// TIA Portal V17 export
// export: Created 2024-08-26T21:10:48.0587448Z, ExportSetting WithDefaults, DisplayName Totally Integrated Automation Portal, DisplayVersion V17 Update 7, DisplayName TIA Portal Openness, DisplayVersion V17 Update 7, DisplayName TIA Portal Version Control Interface, DisplayVersion V17, DisplayName SINAMICS Startdrive Advanced, DisplayVersion V17 SP2, DisplayName SINAMICS Startdrive G110M, G120, G120C, G120D, G120P, G115D, DisplayVersion V17 SP2, DisplayName SINAMICS Startdrive G130, G150, S120, S150, SINAMICS MV, S210, DisplayVersion V17 SP2, DisplayName STEP 7 Professional, DisplayVersion V17 Update 7, DisplayName STEP 7 Safety, DisplayVersion V17 Update 6, DisplayName WinCC Advanced / Unified PC, DisplayVersion V17 Update 7
FUNCTION "outputsMapping" : Void   // FC8, LAD
{ S7_Optimized_Access := 'TRUE' }
VERSION : 0.1
// stored: AutoNumber true, IsIECCheckEnabled false, SetENOAutomatically false, UDAEnableTagReadback false
BEGIN

REGION Network 1: OUTPUT VALVE ACTIVATION
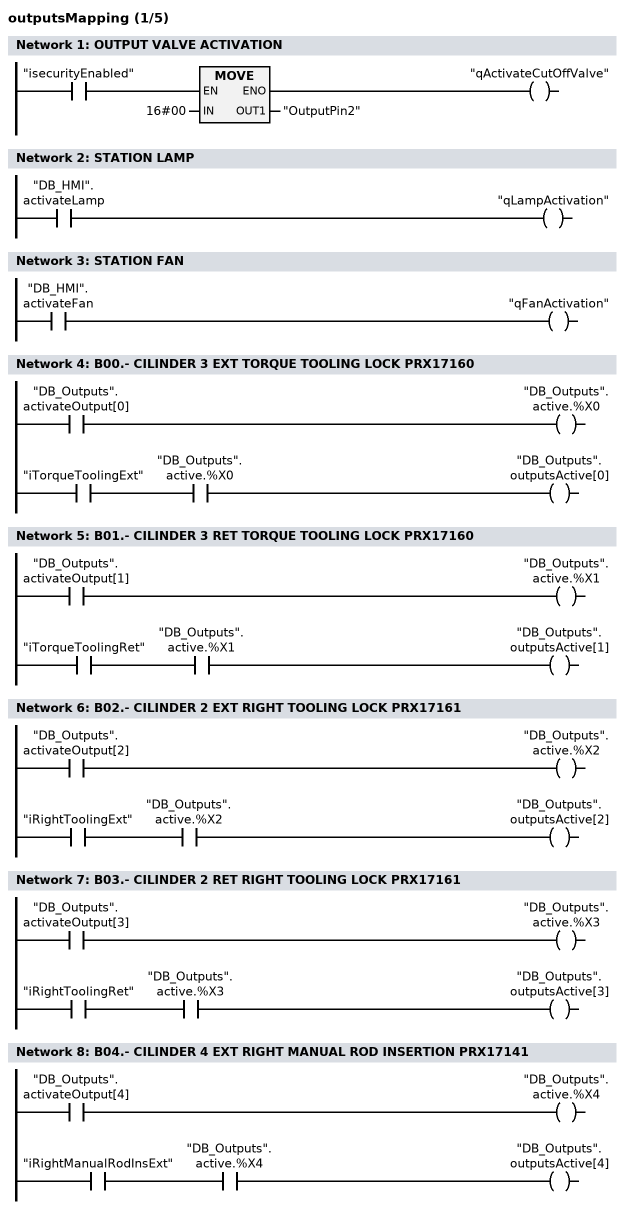
   RUNG wire#powerrail
      Contact( "isecurityEnabled" )
      Move(in := 16#00, out1 => "OutputPin2")
      Coil( "qActivateCutOffValve" )
   END_RUNG
   // the same network as SCL:
   IF "isecurityEnabled" THEN "OutputPin2" := 16#00; END_IF;
   "qActivateCutOffValve" := "isecurityEnabled";
END_REGION

REGION Network 2: STATION LAMP
   RUNG wire#powerrail
      Contact( "DB_HMI".activateLamp )
      Coil( "qLampActivation" )
   END_RUNG
   // the same network as SCL:
   "qLampActivation" := "DB_HMI".activateLamp;
END_REGION

REGION Network 3: STATION FAN
   RUNG wire#powerrail
      Contact( "DB_HMI".activateFan )
      Coil( "qFanActivation" )
   END_RUNG
   // the same network as SCL:
   "qFanActivation" := "DB_HMI".activateFan;
END_REGION

REGION Network 4: B00.- CILINDER 3 EXT TORQUE TOOLING LOCK PRX17160
   RUNG wire#powerrail
      Contact( "DB_Outputs".activateOutput[0] )
      Coil( "DB_Outputs".active.%X0 )
   END_RUNG
   RUNG wire#powerrail
      Contact( "iTorqueToolingExt" )
      Contact( "DB_Outputs".active.%X0 )
      Coil( "DB_Outputs".outputsActive[0] )
   END_RUNG
   // the same network as SCL:
   "DB_Outputs".active.%X0 := "DB_Outputs".activateOutput[0];
   "DB_Outputs".outputsActive[0] := "iTorqueToolingExt" AND "DB_Outputs".active.%X0;
END_REGION

REGION Network 5: B01.- CILINDER 3 RET TORQUE TOOLING LOCK PRX17160
   RUNG wire#powerrail
      Contact( "DB_Outputs".activateOutput[1] )
      Coil( "DB_Outputs".active.%X1 )
   END_RUNG
   RUNG wire#powerrail
      Contact( "iTorqueToolingRet" )
      Contact( "DB_Outputs".active.%X1 )
      Coil( "DB_Outputs".outputsActive[1] )
   END_RUNG
   // the same network as SCL:
   "DB_Outputs".active.%X1 := "DB_Outputs".activateOutput[1];
   "DB_Outputs".outputsActive[1] := "iTorqueToolingRet" AND "DB_Outputs".active.%X1;
END_REGION

REGION Network 6: B02.- CILINDER 2 EXT RIGHT TOOLING LOCK PRX17161
   RUNG wire#powerrail
      Contact( "DB_Outputs".activateOutput[2] )
      Coil( "DB_Outputs".active.%X2 )
   END_RUNG
   RUNG wire#powerrail
      Contact( "iRightToolingExt" )
      Contact( "DB_Outputs".active.%X2 )
      Coil( "DB_Outputs".outputsActive[2] )
   END_RUNG
   // the same network as SCL:
   "DB_Outputs".active.%X2 := "DB_Outputs".activateOutput[2];
   "DB_Outputs".outputsActive[2] := "iRightToolingExt" AND "DB_Outputs".active.%X2;
END_REGION

REGION Network 7: B03.- CILINDER 2 RET RIGHT TOOLING LOCK PRX17161
   RUNG wire#powerrail
      Contact( "DB_Outputs".activateOutput[3] )
      Coil( "DB_Outputs".active.%X3 )
   END_RUNG
   RUNG wire#powerrail
      Contact( "iRightToolingRet" )
      Contact( "DB_Outputs".active.%X3 )
      Coil( "DB_Outputs".outputsActive[3] )
   END_RUNG
   // the same network as SCL:
   "DB_Outputs".active.%X3 := "DB_Outputs".activateOutput[3];
   "DB_Outputs".outputsActive[3] := "iRightToolingRet" AND "DB_Outputs".active.%X3;
END_REGION

REGION Network 8: B04.- CILINDER 4 EXT RIGHT MANUAL ROD INSERTION PRX17141
   RUNG wire#powerrail
      Contact( "DB_Outputs".activateOutput[4] )
      Coil( "DB_Outputs".active.%X4 )
   END_RUNG
   RUNG wire#powerrail
      Contact( "iRightManualRodInsExt" )
      Contact( "DB_Outputs".active.%X4 )
      Coil( "DB_Outputs".outputsActive[4] )
   END_RUNG
   // the same network as SCL:
   "DB_Outputs".active.%X4 := "DB_Outputs".activateOutput[4];
   "DB_Outputs".outputsActive[4] := "iRightManualRodInsExt" AND "DB_Outputs".active.%X4;
END_REGION

REGION Network 9: B05.- CILINDER 4 RET RIGHT MANUAL ROD INSERTION PRX17141
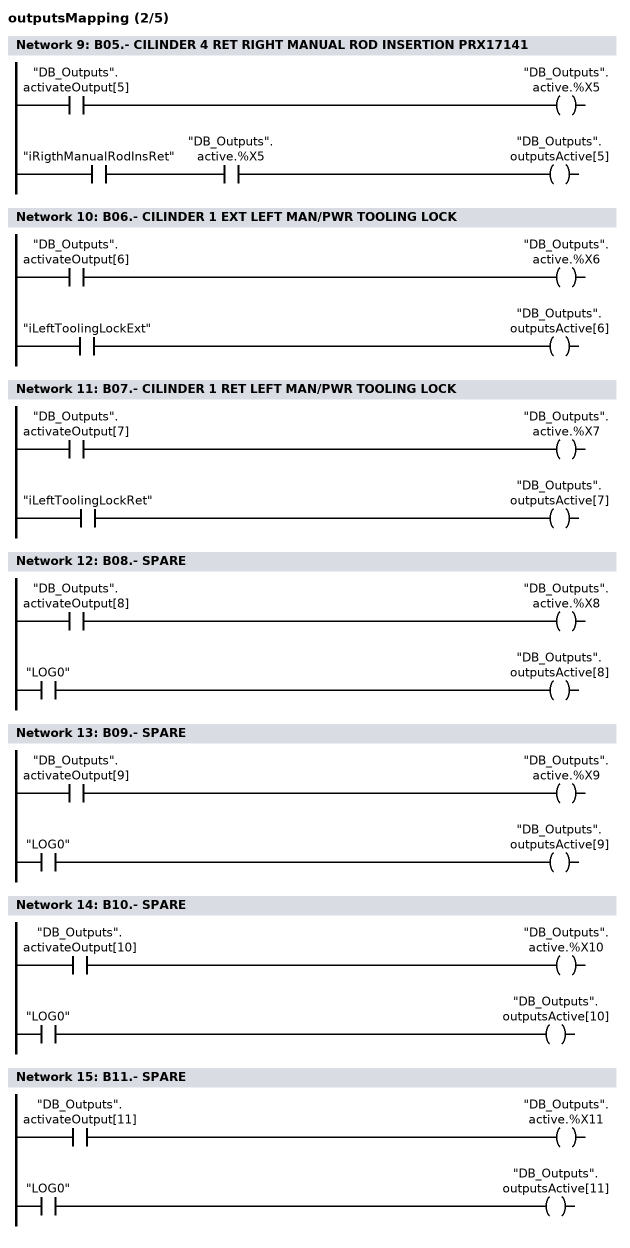
   RUNG wire#powerrail
      Contact( "DB_Outputs".activateOutput[5] )
      Coil( "DB_Outputs".active.%X5 )
   END_RUNG
   RUNG wire#powerrail
      Contact( "iRigthManualRodInsRet" )
      Contact( "DB_Outputs".active.%X5 )
      Coil( "DB_Outputs".outputsActive[5] )
   END_RUNG
   // the same network as SCL:
   "DB_Outputs".active.%X5 := "DB_Outputs".activateOutput[5];
   "DB_Outputs".outputsActive[5] := "iRigthManualRodInsRet" AND "DB_Outputs".active.%X5;
END_REGION

REGION Network 10: B06.- CILINDER 1 EXT LEFT MAN/PWR TOOLING LOCK
   RUNG wire#powerrail
      Contact( "DB_Outputs".activateOutput[6] )
      Coil( "DB_Outputs".active.%X6 )
   END_RUNG
   RUNG wire#powerrail
      Contact( "iLeftToolingLockExt" )
      Coil( "DB_Outputs".outputsActive[6] )
   END_RUNG
   // the same network as SCL:
   "DB_Outputs".active.%X6 := "DB_Outputs".activateOutput[6];
   "DB_Outputs".outputsActive[6] := "iLeftToolingLockExt";
END_REGION

REGION Network 11: B07.- CILINDER 1 RET LEFT MAN/PWR TOOLING LOCK
   RUNG wire#powerrail
      Contact( "DB_Outputs".activateOutput[7] )
      Coil( "DB_Outputs".active.%X7 )
   END_RUNG
   RUNG wire#powerrail
      Contact( "iLeftToolingLockRet" )
      Coil( "DB_Outputs".outputsActive[7] )
   END_RUNG
   // the same network as SCL:
   "DB_Outputs".active.%X7 := "DB_Outputs".activateOutput[7];
   "DB_Outputs".outputsActive[7] := "iLeftToolingLockRet";
END_REGION

REGION Network 12: B08.- SPARE
   RUNG wire#powerrail
      Contact( "DB_Outputs".activateOutput[8] )
      Coil( "DB_Outputs".active.%X8 )
   END_RUNG
   RUNG wire#powerrail
      Contact( "LOG0" )
      Coil( "DB_Outputs".outputsActive[8] )
   END_RUNG
   // the same network as SCL:
   "DB_Outputs".active.%X8 := "DB_Outputs".activateOutput[8];
   "DB_Outputs".outputsActive[8] := "LOG0";
END_REGION

REGION Network 13: B09.- SPARE
   RUNG wire#powerrail
      Contact( "DB_Outputs".activateOutput[9] )
      Coil( "DB_Outputs".active.%X9 )
   END_RUNG
   RUNG wire#powerrail
      Contact( "LOG0" )
      Coil( "DB_Outputs".outputsActive[9] )
   END_RUNG
   // the same network as SCL:
   "DB_Outputs".active.%X9 := "DB_Outputs".activateOutput[9];
   "DB_Outputs".outputsActive[9] := "LOG0";
END_REGION

REGION Network 14: B10.- SPARE
   RUNG wire#powerrail
      Contact( "DB_Outputs".activateOutput[10] )
      Coil( "DB_Outputs".active.%X10 )
   END_RUNG
   RUNG wire#powerrail
      Contact( "LOG0" )
      Coil( "DB_Outputs".outputsActive[10] )
   END_RUNG
   // the same network as SCL:
   "DB_Outputs".active.%X10 := "DB_Outputs".activateOutput[10];
   "DB_Outputs".outputsActive[10] := "LOG0";
END_REGION

REGION Network 15: B11.- SPARE
   RUNG wire#powerrail
      Contact( "DB_Outputs".activateOutput[11] )
      Coil( "DB_Outputs".active.%X11 )
   END_RUNG
   RUNG wire#powerrail
      Contact( "LOG0" )
      Coil( "DB_Outputs".outputsActive[11] )
   END_RUNG
   // the same network as SCL:
   "DB_Outputs".active.%X11 := "DB_Outputs".activateOutput[11];
   "DB_Outputs".outputsActive[11] := "LOG0";
END_REGION

REGION Network 16: B12.- CILINDER 7 EXT INSERTION CYLINDERS WASHER/ROD
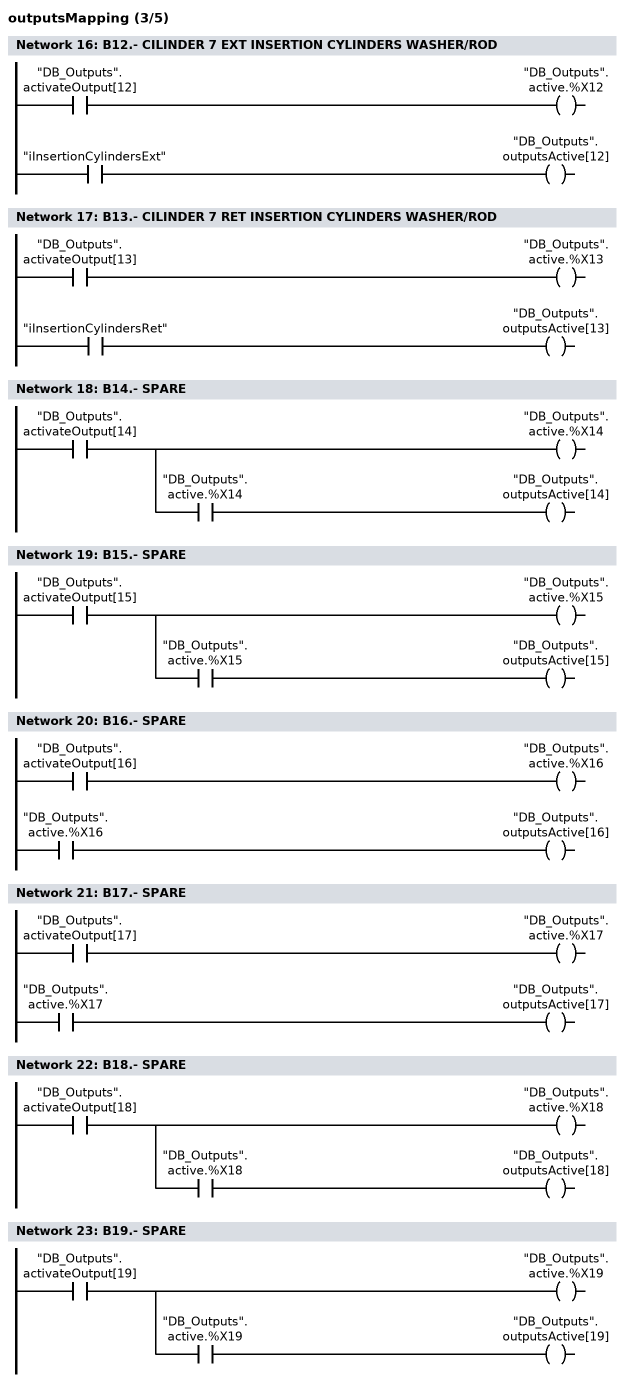
   RUNG wire#powerrail
      Contact( "DB_Outputs".activateOutput[12] )
      Coil( "DB_Outputs".active.%X12 )
   END_RUNG
   RUNG wire#powerrail
      Contact( "iInsertionCylindersExt" )
      Coil( "DB_Outputs".outputsActive[12] )
   END_RUNG
   // the same network as SCL:
   "DB_Outputs".active.%X12 := "DB_Outputs".activateOutput[12];
   "DB_Outputs".outputsActive[12] := "iInsertionCylindersExt";
END_REGION

REGION Network 17: B13.- CILINDER 7 RET INSERTION CYLINDERS WASHER/ROD
   RUNG wire#powerrail
      Contact( "DB_Outputs".activateOutput[13] )
      Coil( "DB_Outputs".active.%X13 )
   END_RUNG
   RUNG wire#powerrail
      Contact( "iInsertionCylindersRet" )
      Coil( "DB_Outputs".outputsActive[13] )
   END_RUNG
   // the same network as SCL:
   "DB_Outputs".active.%X13 := "DB_Outputs".activateOutput[13];
   "DB_Outputs".outputsActive[13] := "iInsertionCylindersRet";
END_REGION

REGION Network 18: B14.- SPARE
   RUNG wire#powerrail
      Contact( "DB_Outputs".activateOutput[14] )
      wire#w1
      Coil( "DB_Outputs".active.%X14 )
   END_RUNG
   RUNG wire#w1
      Contact( "DB_Outputs".active.%X14 )
      Coil( "DB_Outputs".outputsActive[14] )
   END_RUNG
   // the same network as SCL:
   "DB_Outputs".active.%X14 := "DB_Outputs".activateOutput[14];
   "DB_Outputs".outputsActive[14] := "DB_Outputs".activateOutput[14] AND "DB_Outputs".active.%X14;
END_REGION

REGION Network 19: B15.- SPARE
   RUNG wire#powerrail
      Contact( "DB_Outputs".activateOutput[15] )
      wire#w1
      Coil( "DB_Outputs".active.%X15 )
   END_RUNG
   RUNG wire#w1
      Contact( "DB_Outputs".active.%X15 )
      Coil( "DB_Outputs".outputsActive[15] )
   END_RUNG
   // the same network as SCL:
   "DB_Outputs".active.%X15 := "DB_Outputs".activateOutput[15];
   "DB_Outputs".outputsActive[15] := "DB_Outputs".activateOutput[15] AND "DB_Outputs".active.%X15;
END_REGION

REGION Network 20: B16.- SPARE
   RUNG wire#powerrail
      Contact( "DB_Outputs".activateOutput[16] )
      Coil( "DB_Outputs".active.%X16 )
   END_RUNG
   RUNG wire#powerrail
      Contact( "DB_Outputs".active.%X16 )
      Coil( "DB_Outputs".outputsActive[16] )
   END_RUNG
   // the same network as SCL:
   "DB_Outputs".active.%X16 := "DB_Outputs".activateOutput[16];
   "DB_Outputs".outputsActive[16] := "DB_Outputs".active.%X16;
END_REGION

REGION Network 21: B17.- SPARE
   RUNG wire#powerrail
      Contact( "DB_Outputs".activateOutput[17] )
      Coil( "DB_Outputs".active.%X17 )
   END_RUNG
   RUNG wire#powerrail
      Contact( "DB_Outputs".active.%X17 )
      Coil( "DB_Outputs".outputsActive[17] )
   END_RUNG
   // the same network as SCL:
   "DB_Outputs".active.%X17 := "DB_Outputs".activateOutput[17];
   "DB_Outputs".outputsActive[17] := "DB_Outputs".active.%X17;
END_REGION

REGION Network 22: B18.- SPARE
   RUNG wire#powerrail
      Contact( "DB_Outputs".activateOutput[18] )
      wire#w1
      Coil( "DB_Outputs".active.%X18 )
   END_RUNG
   RUNG wire#w1
      Contact( "DB_Outputs".active.%X18 )
      Coil( "DB_Outputs".outputsActive[18] )
   END_RUNG
   // the same network as SCL:
   "DB_Outputs".active.%X18 := "DB_Outputs".activateOutput[18];
   "DB_Outputs".outputsActive[18] := "DB_Outputs".activateOutput[18] AND "DB_Outputs".active.%X18;
END_REGION

REGION Network 23: B19.- SPARE
   RUNG wire#powerrail
      Contact( "DB_Outputs".activateOutput[19] )
      wire#w1
      Coil( "DB_Outputs".active.%X19 )
   END_RUNG
   RUNG wire#w1
      Contact( "DB_Outputs".active.%X19 )
      Coil( "DB_Outputs".outputsActive[19] )
   END_RUNG
   // the same network as SCL:
   "DB_Outputs".active.%X19 := "DB_Outputs".activateOutput[19];
   "DB_Outputs".outputsActive[19] := "DB_Outputs".activateOutput[19] AND "DB_Outputs".active.%X19;
END_REGION

REGION Network 24: B20.- SPARE
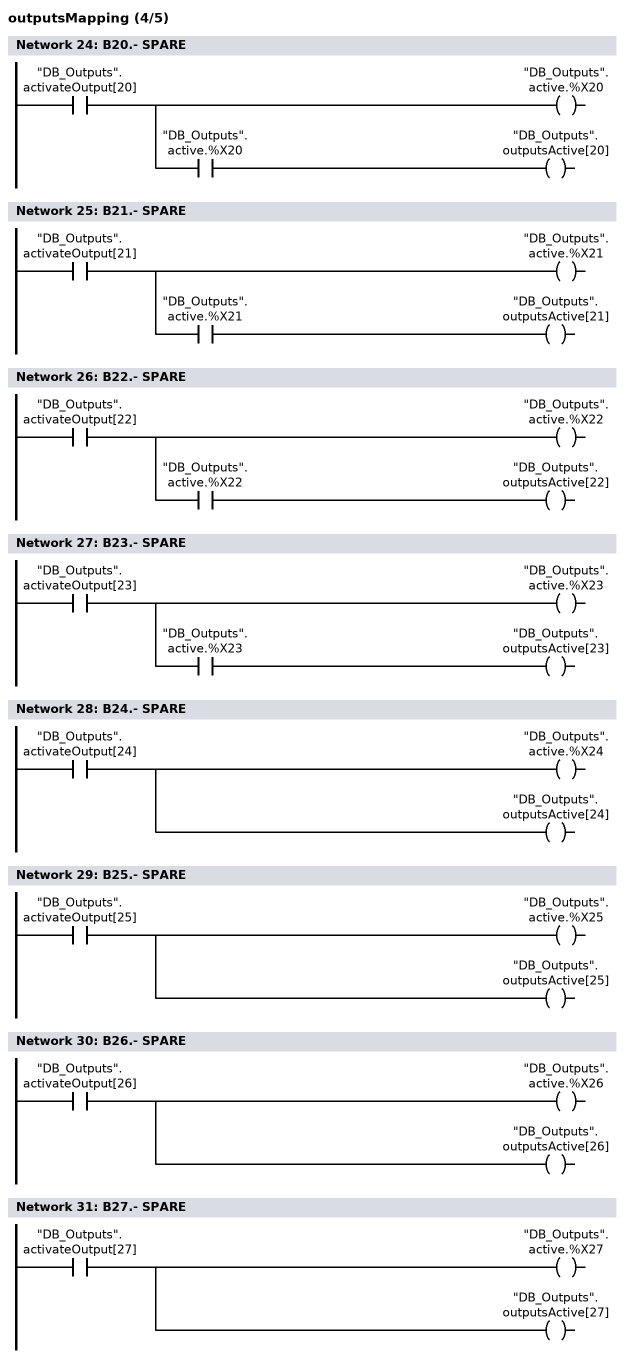
   RUNG wire#powerrail
      Contact( "DB_Outputs".activateOutput[20] )
      wire#w1
      Coil( "DB_Outputs".active.%X20 )
   END_RUNG
   RUNG wire#w1
      Contact( "DB_Outputs".active.%X20 )
      Coil( "DB_Outputs".outputsActive[20] )
   END_RUNG
   // the same network as SCL:
   "DB_Outputs".active.%X20 := "DB_Outputs".activateOutput[20];
   "DB_Outputs".outputsActive[20] := "DB_Outputs".activateOutput[20] AND "DB_Outputs".active.%X20;
END_REGION

REGION Network 25: B21.- SPARE
   RUNG wire#powerrail
      Contact( "DB_Outputs".activateOutput[21] )
      wire#w1
      Coil( "DB_Outputs".active.%X21 )
   END_RUNG
   RUNG wire#w1
      Contact( "DB_Outputs".active.%X21 )
      Coil( "DB_Outputs".outputsActive[21] )
   END_RUNG
   // the same network as SCL:
   "DB_Outputs".active.%X21 := "DB_Outputs".activateOutput[21];
   "DB_Outputs".outputsActive[21] := "DB_Outputs".activateOutput[21] AND "DB_Outputs".active.%X21;
END_REGION

REGION Network 26: B22.- SPARE
   RUNG wire#powerrail
      Contact( "DB_Outputs".activateOutput[22] )
      wire#w1
      Coil( "DB_Outputs".active.%X22 )
   END_RUNG
   RUNG wire#w1
      Contact( "DB_Outputs".active.%X22 )
      Coil( "DB_Outputs".outputsActive[22] )
   END_RUNG
   // the same network as SCL:
   "DB_Outputs".active.%X22 := "DB_Outputs".activateOutput[22];
   "DB_Outputs".outputsActive[22] := "DB_Outputs".activateOutput[22] AND "DB_Outputs".active.%X22;
END_REGION

REGION Network 27: B23.- SPARE
   RUNG wire#powerrail
      Contact( "DB_Outputs".activateOutput[23] )
      wire#w1
      Coil( "DB_Outputs".active.%X23 )
   END_RUNG
   RUNG wire#w1
      Contact( "DB_Outputs".active.%X23 )
      Coil( "DB_Outputs".outputsActive[23] )
   END_RUNG
   // the same network as SCL:
   "DB_Outputs".active.%X23 := "DB_Outputs".activateOutput[23];
   "DB_Outputs".outputsActive[23] := "DB_Outputs".activateOutput[23] AND "DB_Outputs".active.%X23;
END_REGION

REGION Network 28: B24.- SPARE
   RUNG wire#powerrail
      Contact( "DB_Outputs".activateOutput[24] )
      wire#w1
      Coil( "DB_Outputs".active.%X24 )
   END_RUNG
   RUNG wire#w1
      Coil( "DB_Outputs".outputsActive[24] )
   END_RUNG
   // the same network as SCL:
   "DB_Outputs".active.%X24 := "DB_Outputs".activateOutput[24];
   "DB_Outputs".outputsActive[24] := "DB_Outputs".activateOutput[24];
END_REGION

REGION Network 29: B25.- SPARE
   RUNG wire#powerrail
      Contact( "DB_Outputs".activateOutput[25] )
      wire#w1
      Coil( "DB_Outputs".active.%X25 )
   END_RUNG
   RUNG wire#w1
      Coil( "DB_Outputs".outputsActive[25] )
   END_RUNG
   // the same network as SCL:
   "DB_Outputs".active.%X25 := "DB_Outputs".activateOutput[25];
   "DB_Outputs".outputsActive[25] := "DB_Outputs".activateOutput[25];
END_REGION

REGION Network 30: B26.- SPARE
   RUNG wire#powerrail
      Contact( "DB_Outputs".activateOutput[26] )
      wire#w1
      Coil( "DB_Outputs".active.%X26 )
   END_RUNG
   RUNG wire#w1
      Coil( "DB_Outputs".outputsActive[26] )
   END_RUNG
   // the same network as SCL:
   "DB_Outputs".active.%X26 := "DB_Outputs".activateOutput[26];
   "DB_Outputs".outputsActive[26] := "DB_Outputs".activateOutput[26];
END_REGION

REGION Network 31: B27.- SPARE
   RUNG wire#powerrail
      Contact( "DB_Outputs".activateOutput[27] )
      wire#w1
      Coil( "DB_Outputs".active.%X27 )
   END_RUNG
   RUNG wire#w1
      Coil( "DB_Outputs".outputsActive[27] )
   END_RUNG
   // the same network as SCL:
   "DB_Outputs".active.%X27 := "DB_Outputs".activateOutput[27];
   "DB_Outputs".outputsActive[27] := "DB_Outputs".activateOutput[27];
END_REGION

REGION Network 32: B28.- SPARE
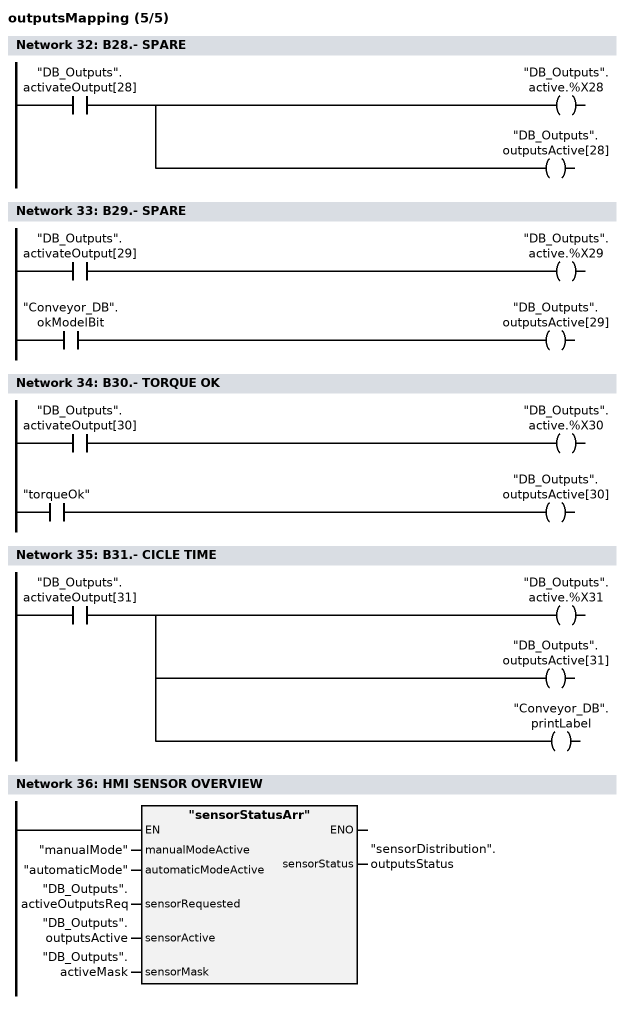
   RUNG wire#powerrail
      Contact( "DB_Outputs".activateOutput[28] )
      wire#w1
      Coil( "DB_Outputs".active.%X28 )
   END_RUNG
   RUNG wire#w1
      Coil( "DB_Outputs".outputsActive[28] )
   END_RUNG
   // the same network as SCL:
   "DB_Outputs".active.%X28 := "DB_Outputs".activateOutput[28];
   "DB_Outputs".outputsActive[28] := "DB_Outputs".activateOutput[28];
END_REGION

REGION Network 33: B29.- SPARE
   RUNG wire#powerrail
      Contact( "DB_Outputs".activateOutput[29] )
      Coil( "DB_Outputs".active.%X29 )
   END_RUNG
   RUNG wire#powerrail
      Contact( "Conveyor_DB".okModelBit )
      Coil( "DB_Outputs".outputsActive[29] )
   END_RUNG
   // the same network as SCL:
   "DB_Outputs".active.%X29 := "DB_Outputs".activateOutput[29];
   "DB_Outputs".outputsActive[29] := "Conveyor_DB".okModelBit;
END_REGION

REGION Network 34: B30.- TORQUE OK
   RUNG wire#powerrail
      Contact( "DB_Outputs".activateOutput[30] )
      Coil( "DB_Outputs".active.%X30 )
   END_RUNG
   RUNG wire#powerrail
      Contact( "torqueOk" )
      Coil( "DB_Outputs".outputsActive[30] )
   END_RUNG
   // the same network as SCL:
   "DB_Outputs".active.%X30 := "DB_Outputs".activateOutput[30];
   "DB_Outputs".outputsActive[30] := "torqueOk";
END_REGION

REGION Network 35: B31.- CICLE TIME
   RUNG wire#powerrail
      Contact( "DB_Outputs".activateOutput[31] )
      wire#w1
      Coil( "DB_Outputs".active.%X31 )
   END_RUNG
   RUNG wire#w1
      Coil( "DB_Outputs".outputsActive[31] )
   END_RUNG
   RUNG wire#w1
      Coil( "Conveyor_DB".printLabel )
   END_RUNG
   // the same network as SCL:
   "DB_Outputs".active.%X31 := "DB_Outputs".activateOutput[31];
   "DB_Outputs".outputsActive[31] := "DB_Outputs".activateOutput[31];
   "Conveyor_DB".printLabel := "DB_Outputs".activateOutput[31];
END_REGION

REGION Network 36: HMI SENSOR OVERVIEW
   RUNG wire#powerrail
      "sensorStatusArr"(manualModeActive := "manualMode", automaticModeActive := "automaticMode", sensorRequested := "DB_Outputs".activeOutputsReq, sensorActive := "DB_Outputs".outputsActive, sensorMask := "DB_Outputs".activeMask, sensorStatus => "sensorDistribution".outputsStatus)
   END_RUNG
   // the same network as SCL:
   "sensorStatusArr"(manualModeActive := "manualMode",
                     automaticModeActive := "automaticMode",
                     sensorRequested := "DB_Outputs".activeOutputsReq,
                     sensorActive := "DB_Outputs".outputsActive,
                     sensorMask := "DB_Outputs".activeMask,
                     sensorStatus => "sensorDistribution".outputsStatus);
END_REGION
END_FUNCTION
